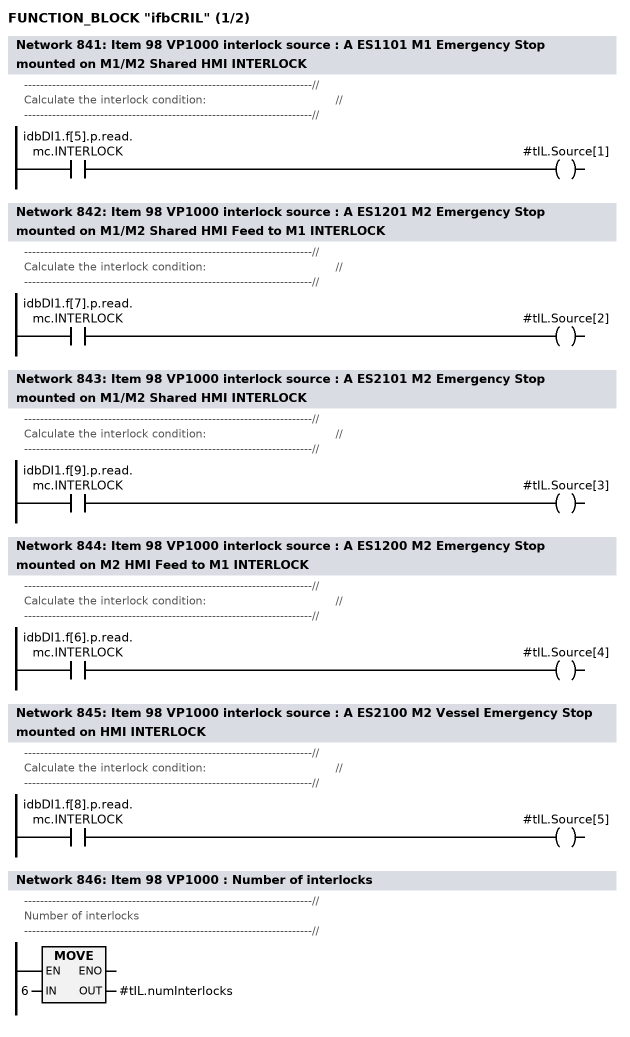
    A idbDI1.f[5].p.read.mc.INTERLOCK;
    = #tIL.Source[1];

NETWORK
TITLE = Item 98 VP1000 interlock source : A ES1201 M2 Emergency Stop mounted on M1/M2 Shared HMI Feed to M1 INTERLOCK
    //------------------------------------------------------------------------//
    // Calculate the interlock condition:                                     //
    //------------------------------------------------------------------------//
    A idbDI1.f[7].p.read.mc.INTERLOCK;
    = #tIL.Source[2];

NETWORK
TITLE = Item 98 VP1000 interlock source : A ES2101 M2 Emergency Stop mounted on M1/M2 Shared HMI INTERLOCK
    //------------------------------------------------------------------------//
    // Calculate the interlock condition:                                     //
    //------------------------------------------------------------------------//
    A idbDI1.f[9].p.read.mc.INTERLOCK;
    = #tIL.Source[3];

NETWORK
TITLE = Item 98 VP1000 interlock source : A ES1200 M2 Emergency Stop mounted on M2 HMI Feed to M1 INTERLOCK
    //------------------------------------------------------------------------//
    // Calculate the interlock condition:                                     //
    //------------------------------------------------------------------------//
    A idbDI1.f[6].p.read.mc.INTERLOCK;
    = #tIL.Source[4];

NETWORK
TITLE = Item 98 VP1000 interlock source : A ES2100 M2 Vessel Emergency Stop mounted on HMI INTERLOCK
    //------------------------------------------------------------------------//
    // Calculate the interlock condition:                                     //
    //------------------------------------------------------------------------//
    A idbDI1.f[8].p.read.mc.INTERLOCK;
    = #tIL.Source[5];


NETWORK
TITLE = Item 98 VP1000 : Number of interlocks
    //------------------------------------------------------------------------//
    // Number of interlocks
    //------------------------------------------------------------------------//
    L 6;
    T #tIL.numInterlocks;

NETWORK
TITLE = Item 98 VP1000 : Aggregate individual interlocks into overall INTERLOCK flag
    //------------------------------------------------------------------------//
    // Determine if an interlock is raised:                                   //
    //------------------------------------------------------------------------//
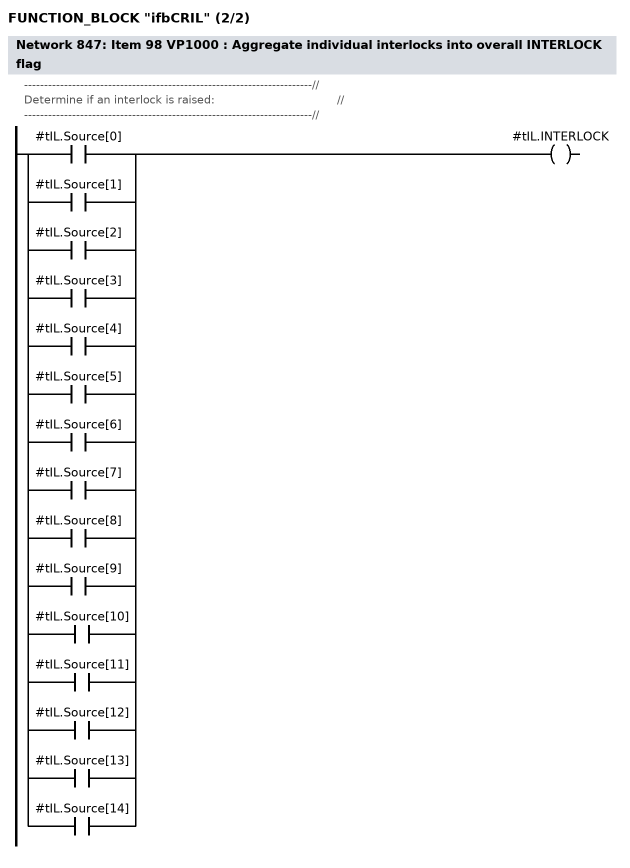
    O #tIL.Source[0];
    O #tIL.Source[1];
    O #tIL.Source[2];
    O #tIL.Source[3];
    O #tIL.Source[4];
    O #tIL.Source[5];
    O #tIL.Source[6];
    O #tIL.Source[7];
    O #tIL.Source[8];
    O #tIL.Source[9];
    O #tIL.Source[10];
    O #tIL.Source[11];
    O #tIL.Source[12];
    O #tIL.Source[13];
    O #tIL.Source[14];
    = #tIL.INTERLOCK;

NETWORK
TITLE = Item 98 VP1000 : Update the instance data
    //------------------------------------------------------------------------//
    // Update the instance DB with the calculated interlock flags:            //
    //------------------------------------------------------------------------//
    CALL MOVE
    {value_type := 'Variant'}
    (   IN                   := #tIL ,
        OUT                  := #p[98]
    );

NETWORK
TITLE = Item 99 VP1001 : MX Vacuum Pump 2 initialise variables
    //------------------------------------------------------------------------//
    // CRITICAL INTERLOCK   CRITICAL INTERLOCK   CRITICAL INTERLOCK   CRITICA //
    // CRITICAL INTERLOCK   CRITICAL INTERLOCK   CRITICAL INTERLOCK   CRITICA //
    //                                                                        //
    // Clear the interlock flag:                                              //
    //------------------------------------------------------------------------//
    A "alwaysLow";
    = #tIL.INTERLOCK;

    //------------------------------------------------------------------------//
    // Clear all interlock values to initialise them to off:                  //
    //------------------------------------------------------------------------//
    CALL FILL_BLK
    {value_type := 'Bool', count_type := 'UInt'}
    (   IN                   := 0 ,
        COUNT                := 15 ,
        OUT                  := #tIL.Source[0]
    );


NETWORK
TITLE = Item 99 VP1001 interlock source : A ES1100 M1 Vessel Emergency Stop mounted on HMI INTERLOCK
    //------------------------------------------------------------------------//
    // Calculate the interlock condition:                                     //
    //------------------------------------------------------------------------//
    A idbDI1.f[4].p.read.mc.INTERLOCK;
    = #tIL.Source[0];

NETWORK
TITLE = Item 99 VP1001 interlock source : A ES1101 M1 Emergency Stop mounted on M1/M2 Shared HMI INTERLOCK
    //------------------------------------------------------------------------//
    // Calculate the interlock condition:                                     //
    //------------------------------------------------------------------------//
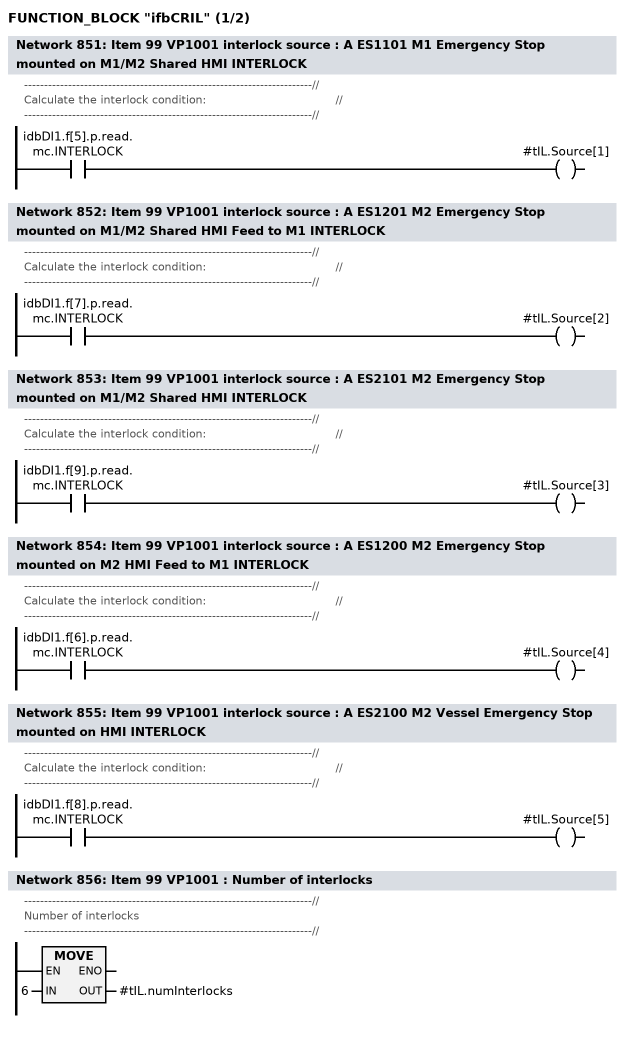
    A idbDI1.f[5].p.read.mc.INTERLOCK;
    = #tIL.Source[1];

NETWORK
TITLE = Item 99 VP1001 interlock source : A ES1201 M2 Emergency Stop mounted on M1/M2 Shared HMI Feed to M1 INTERLOCK
    //------------------------------------------------------------------------//
    // Calculate the interlock condition:                                     //
    //------------------------------------------------------------------------//
    A idbDI1.f[7].p.read.mc.INTERLOCK;
    = #tIL.Source[2];

NETWORK
TITLE = Item 99 VP1001 interlock source : A ES2101 M2 Emergency Stop mounted on M1/M2 Shared HMI INTERLOCK
    //------------------------------------------------------------------------//
    // Calculate the interlock condition:                                     //
    //------------------------------------------------------------------------//
    A idbDI1.f[9].p.read.mc.INTERLOCK;
    = #tIL.Source[3];

NETWORK
TITLE = Item 99 VP1001 interlock source : A ES1200 M2 Emergency Stop mounted on M2 HMI Feed to M1 INTERLOCK
    //------------------------------------------------------------------------//
    // Calculate the interlock condition:                                     //
    //------------------------------------------------------------------------//
    A idbDI1.f[6].p.read.mc.INTERLOCK;
    = #tIL.Source[4];

NETWORK
TITLE = Item 99 VP1001 interlock source : A ES2100 M2 Vessel Emergency Stop mounted on HMI INTERLOCK
    //------------------------------------------------------------------------//
    // Calculate the interlock condition:                                     //
    //------------------------------------------------------------------------//
    A idbDI1.f[8].p.read.mc.INTERLOCK;
    = #tIL.Source[5];


NETWORK
TITLE = Item 99 VP1001 : Number of interlocks
    //------------------------------------------------------------------------//
    // Number of interlocks
    //------------------------------------------------------------------------//
    L 6;
    T #tIL.numInterlocks;

NETWORK
TITLE = Item 99 VP1001 : Aggregate individual interlocks into overall INTERLOCK flag
    //------------------------------------------------------------------------//
    // Determine if an interlock is raised:                                   //
    //------------------------------------------------------------------------//
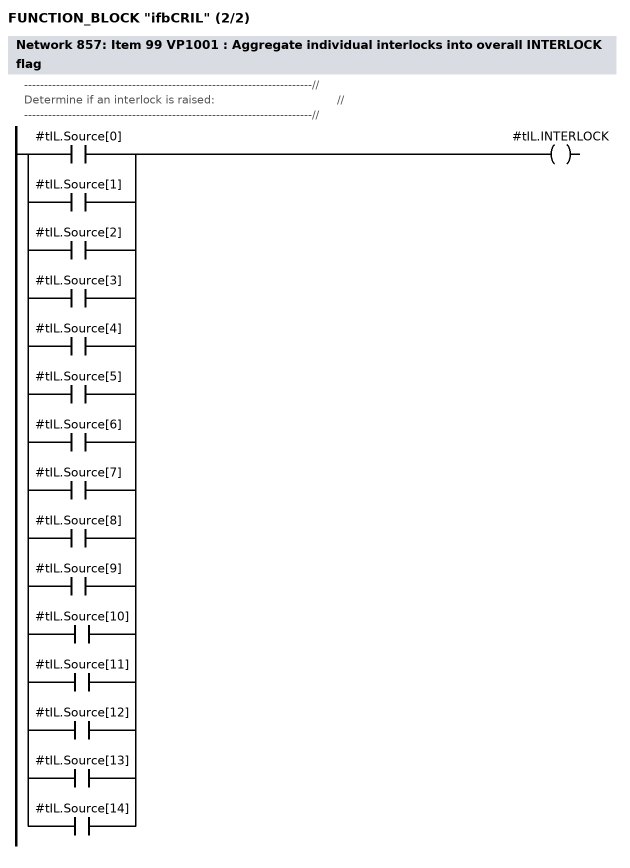
    O #tIL.Source[0];
    O #tIL.Source[1];
    O #tIL.Source[2];
    O #tIL.Source[3];
    O #tIL.Source[4];
    O #tIL.Source[5];
    O #tIL.Source[6];
    O #tIL.Source[7];
    O #tIL.Source[8];
    O #tIL.Source[9];
    O #tIL.Source[10];
    O #tIL.Source[11];
    O #tIL.Source[12];
    O #tIL.Source[13];
    O #tIL.Source[14];
    = #tIL.INTERLOCK;

NETWORK
TITLE = Item 99 VP1001 : Update the instance data
    //------------------------------------------------------------------------//
    // Update the instance DB with the calculated interlock flags:            //
    //------------------------------------------------------------------------//
    CALL MOVE
    {value_type := 'Variant'}
    (   IN                   := #tIL ,
        OUT                  := #p[99]
    );

NETWORK
TITLE = Item 100 VP3000 : SY Vacuum Pump 1 initialise variables
    //------------------------------------------------------------------------//
    // CRITICAL INTERLOCK   CRITICAL INTERLOCK   CRITICAL INTERLOCK   CRITICA //
    // CRITICAL INTERLOCK   CRITICAL INTERLOCK   CRITICAL INTERLOCK   CRITICA //
    //                                                                        //
    // Clear the interlock flag:                                              //
    //------------------------------------------------------------------------//
    A "alwaysLow";
    = #tIL.INTERLOCK;

    //------------------------------------------------------------------------//
    // Clear all interlock values to initialise them to off:                  //
    //------------------------------------------------------------------------//
    CALL FILL_BLK
    {value_type := 'Bool', count_type := 'UInt'}
    (   IN                   := 0 ,
        COUNT                := 15 ,
        OUT                  := #tIL.Source[0]
    );


NETWORK
TITLE = Item 100 VP3000 interlock source : A ES3100 S1 Emergency Stop mounted on S1 HMI INTERLOCK
    //------------------------------------------------------------------------//
    // Calculate the interlock condition:                                     //
    //------------------------------------------------------------------------//
    A idbDI1.f[10].p.read.mc.INTERLOCK;
    = #tIL.Source[0];

NETWORK
TITLE = Item 100 VP3000 interlock source : A ES3400 S2 Emergency Stop mounted on S2 HMI Feed to S1 INTERLOCK
    //------------------------------------------------------------------------//
    // Calculate the interlock condition:                                     //
    //------------------------------------------------------------------------//
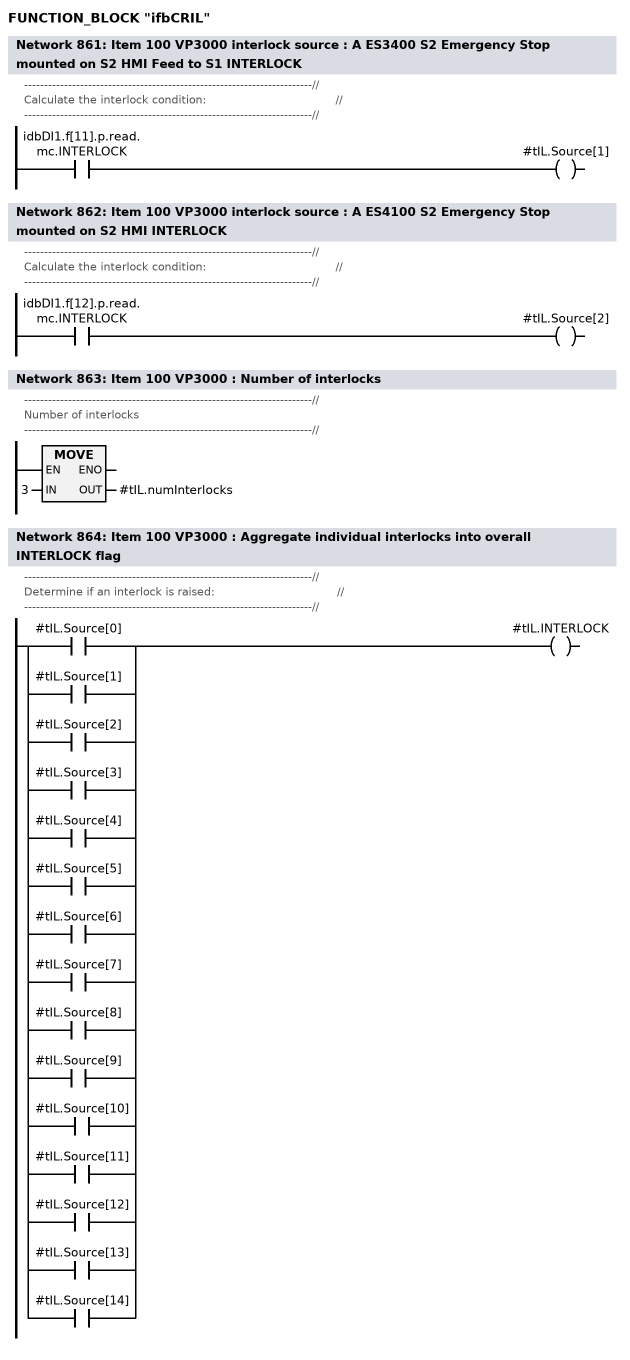
    A idbDI1.f[11].p.read.mc.INTERLOCK;
    = #tIL.Source[1];

NETWORK
TITLE = Item 100 VP3000 interlock source : A ES4100 S2 Emergency Stop mounted on S2 HMI INTERLOCK
    //------------------------------------------------------------------------//
    // Calculate the interlock condition:                                     //
    //------------------------------------------------------------------------//
    A idbDI1.f[12].p.read.mc.INTERLOCK;
    = #tIL.Source[2];


NETWORK
TITLE = Item 100 VP3000 : Number of interlocks
    //------------------------------------------------------------------------//
    // Number of interlocks
    //------------------------------------------------------------------------//
    L 3;
    T #tIL.numInterlocks;

NETWORK
TITLE = Item 100 VP3000 : Aggregate individual interlocks into overall INTERLOCK flag
    //------------------------------------------------------------------------//
    // Determine if an interlock is raised:                                   //
    //------------------------------------------------------------------------//
    O #tIL.Source[0];
    O #tIL.Source[1];
    O #tIL.Source[2];
    O #tIL.Source[3];
    O #tIL.Source[4];
    O #tIL.Source[5];
    O #tIL.Source[6];
    O #tIL.Source[7];
    O #tIL.Source[8];
    O #tIL.Source[9];
    O #tIL.Source[10];
    O #tIL.Source[11];
    O #tIL.Source[12];
    O #tIL.Source[13];
    O #tIL.Source[14];
    = #tIL.INTERLOCK;

NETWORK
TITLE = Item 100 VP3000 : Update the instance data
    //------------------------------------------------------------------------//
    // Update the instance DB with the calculated interlock flags:            //
    //------------------------------------------------------------------------//
    CALL MOVE
    {value_type := 'Variant'}
    (   IN                   := #tIL ,
        OUT                  := #p[100]
    );

NETWORK
TITLE = Item 101 VP3001 : SY Vacuum Pump 2 initialise variables
    //------------------------------------------------------------------------//
    // CRITICAL INTERLOCK   CRITICAL INTERLOCK   CRITICAL INTERLOCK   CRITICA //
    // CRITICAL INTERLOCK   CRITICAL INTERLOCK   CRITICAL INTERLOCK   CRITICA //
    //                                                                        //
    // Clear the interlock flag:                                              //
    //------------------------------------------------------------------------//
    A "alwaysLow";
    = #tIL.INTERLOCK;

    //------------------------------------------------------------------------//
    // Clear all interlock values to initialise them to off:                  //
    //------------------------------------------------------------------------//
    CALL FILL_BLK
    {value_type := 'Bool', count_type := 'UInt'}
    (   IN                   := 0 ,
        COUNT                := 15 ,
        OUT                  := #tIL.Source[0]
    );


NETWORK
TITLE = Item 101 VP3001 interlock source : A ES3100 S1 Emergency Stop mounted on S1 HMI INTERLOCK
    //------------------------------------------------------------------------//
    // Calculate the interlock condition:                                     //
    //------------------------------------------------------------------------//
    A idbDI1.f[10].p.read.mc.INTERLOCK;
    = #tIL.Source[0];

NETWORK
TITLE = Item 101 VP3001 interlock source : A ES3400 S2 Emergency Stop mounted on S2 HMI Feed to S1 INTERLOCK
    //------------------------------------------------------------------------//
    // Calculate the interlock condition:                                     //
    //------------------------------------------------------------------------//
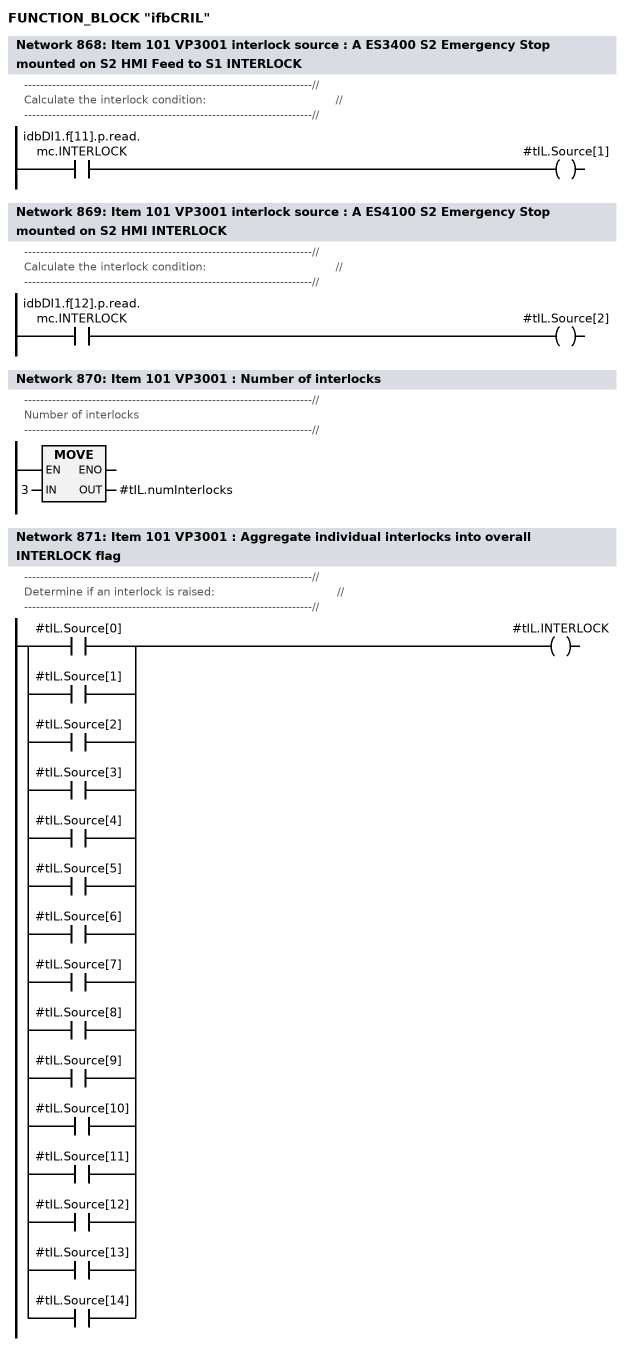
    A idbDI1.f[11].p.read.mc.INTERLOCK;
    = #tIL.Source[1];

NETWORK
TITLE = Item 101 VP3001 interlock source : A ES4100 S2 Emergency Stop mounted on S2 HMI INTERLOCK
    //------------------------------------------------------------------------//
    // Calculate the interlock condition:                                     //
    //------------------------------------------------------------------------//
    A idbDI1.f[12].p.read.mc.INTERLOCK;
    = #tIL.Source[2];


NETWORK
TITLE = Item 101 VP3001 : Number of interlocks
    //------------------------------------------------------------------------//
    // Number of interlocks
    //------------------------------------------------------------------------//
    L 3;
    T #tIL.numInterlocks;

NETWORK
TITLE = Item 101 VP3001 : Aggregate individual interlocks into overall INTERLOCK flag
    //------------------------------------------------------------------------//
    // Determine if an interlock is raised:                                   //
    //------------------------------------------------------------------------//
    O #tIL.Source[0];
    O #tIL.Source[1];
    O #tIL.Source[2];
    O #tIL.Source[3];
    O #tIL.Source[4];
    O #tIL.Source[5];
    O #tIL.Source[6];
    O #tIL.Source[7];
    O #tIL.Source[8];
    O #tIL.Source[9];
    O #tIL.Source[10];
    O #tIL.Source[11];
    O #tIL.Source[12];
    O #tIL.Source[13];
    O #tIL.Source[14];
    = #tIL.INTERLOCK;

NETWORK
TITLE = Item 101 VP3001 : Update the instance data
    //------------------------------------------------------------------------//
    // Update the instance DB with the calculated interlock flags:            //
    //------------------------------------------------------------------------//
    CALL MOVE
    {value_type := 'Variant'}
    (   IN                   := #tIL ,
        OUT                  := #p[101]
    );

END_FUNCTION_BLOCK
